(* IEC 61131-3 sources: RL_MAR/experiments/comparison/autoplc/results/deepseek-ai-DeepSeek-V3.2_20260508_111905/med_81, 1 file *)

(* ---- med_81_1.st ---- *)
FUNCTION_BLOCK SolarPanelTracking
VAR
    PanelAngle : REAL; (* Output for adjusting the solar panel angle *)
    SunriseTime : TIME := T#6H; (* Set the time for sunrise (6:00 AM) *)
    SunsetTime : TIME := T#18H; (* Set the time for sunset (6:00 PM) *)
    NoonTime : TIME := T#12H; (* Set the time for solar noon (12:00 PM) *)
    MorningAngle : REAL := 30.0; (* Set the morning angle for panels *)
    NoonAngle : REAL := 60.0; (* Set the noon angle for panels *)
    EveningAngle : REAL := 30.0; (* Set the evening angle for panels *)
END_VAR
VAR_INPUT
    CurrentTime : TIME;
    SolarIntensity : REAL;
END_VAR

(* Main execution logic *)
IF SolarIntensity >= 90.0 THEN
    (* High-Intensity Override State *)
    PanelAngle := NoonAngle;
ELSE
    (* Time-Based Tracking *)
    IF (CurrentTime < SunriseTime) OR (CurrentTime >= SunsetTime) THEN
        (* Night State *)
        PanelAngle := 0.0;
    ELSIF (CurrentTime >= SunriseTime) AND (CurrentTime < NoonTime) THEN
        (* Morning State *)
        PanelAngle := MorningAngle;
    ELSE
        (* Afternoon/Evening State *)
        PanelAngle := EveningAngle;
    END_IF;
END_IF;

END_FUNCTION_BLOCK
